FUNCTION_BLOCK PnpXYCalculator (* Composite Function Block Type *)
  (* Standard: 61499-2 *)
  (* Version 0.2, 2003-12-05, JHC, Rockwell Automation, Renamed from NEWCOMPFB. *)
  (* Version 0.1, 2002-01-08, JHC, Rockwell Automation, Added DLY FB as example. *)
  (* Version 0.0, 2000-05-27, JHC, Rockwell Automation *)
  (* Compiler header: package fb.rt.pnp; *)
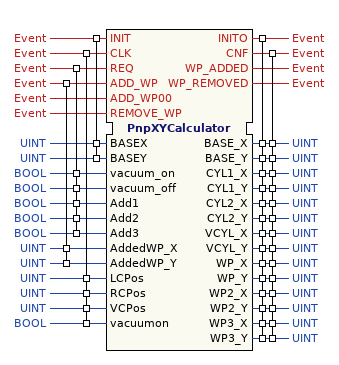
  EVENT_INPUT
    INIT WITH BASEX, BASEY; (* Initialization Request *)
    CLK WITH LCPos, RCPos, VCPos, vacuumon; (* Clock *)
    REQ WITH vacuum_on, vacuum_off, Add1, Add2, Add3;
    ADD_WP WITH AddedWP_X, AddedWP_Y;
    ADD_WP00;
    REMOVE_WP;
  END_EVENT
  EVENT_OUTPUT
    INITO WITH CYL1_X, CYL1_Y, BASE_Y, BASE_X, CYL2_X, CYL2_Y, VCYL_X, VCYL_Y, WP_X, WP_Y, WP2_X, WP2_Y, WP3_X, WP3_Y; (* Initialization Confirm *)
    CNF WITH CYL1_X, CYL1_Y, BASE_Y, BASE_X, CYL2_X, CYL2_Y, VCYL_X, VCYL_Y, WP_X, WP_Y, WP2_X, WP2_Y, WP3_X, WP3_Y;
    WP_ADDED;
    WP_REMOVED;
  END_EVENT
  VAR_INPUT
    BASEX : UINT;
    BASEY : UINT;
    vacuum_on : BOOL;
    vacuum_off : BOOL;
    Add1 : BOOL;
    Add2 : BOOL;
    Add3 : BOOL;
    AddedWP_X : UINT;
    AddedWP_Y : UINT;
    LCPos : UINT;
    RCPos : UINT;
    VCPos : UINT;
    vacuumon : BOOL;
  END_VAR
  VAR_OUTPUT
    BASE_X : UINT; (* Response Data from Socket *)
    BASE_Y : UINT; (* Response Data from Socket *)
    CYL1_X : UINT; (* Response Data from Socket *)
    CYL1_Y : UINT; (* Response Data from Socket *)
    CYL2_X : UINT; (* Response Data from Socket *)
    CYL2_Y : UINT; (* Response Data from Socket *)
    VCYL_X : UINT; (* Response Data from Socket *)
    VCYL_Y : UINT; (* Response Data from Socket *)
    WP_X : UINT; (* Response Data from Socket *)
    WP_Y : UINT; (* Response Data from Socket *)
    WP2_X : UINT; (* Response Data from Socket *)
    WP2_Y : UINT; (* Response Data from Socket *)
    WP3_X : UINT; (* Response Data from Socket *)
    WP3_Y : UINT; (* Response Data from Socket *)
  END_VAR
  VAR
    cyl1x : UINT;
    cyl2x : UINT;
    vcyly : UINT;
    wpx : UINT;
    wpy : UINT;
    wp2x : UINT;
    wp2y : UINT;
    wp3x : UINT;
    wp3y : UINT;
    slider1 : BOOL;
    slider2 : BOOL;
    slider3 : BOOL;
    wpon : BOOL;
    wp2on : BOOL;
    wp3on : BOOL;
  END_VAR
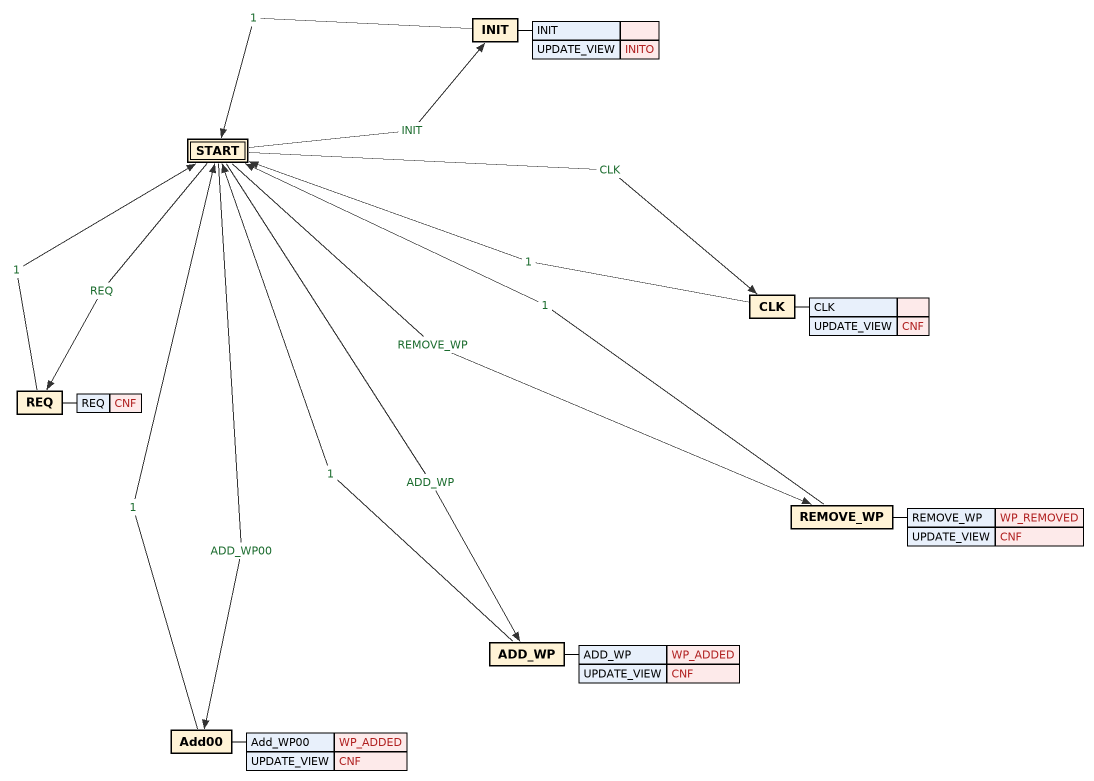
  EC_STATES
    START; (* Initial State *)
    INIT : INIT, UPDATE_VIEW -> INITO; (* Initialization *)
    REQ : REQ -> CNF; (* Normal execution *)
    CLK : CLK, UPDATE_VIEW -> CNF;
    ADD_WP : ADD_WP -> WP_ADDED, UPDATE_VIEW -> CNF;
    REMOVE_WP : REMOVE_WP -> WP_REMOVED, UPDATE_VIEW -> CNF;
    Add00 : Add_WP00 -> WP_ADDED, UPDATE_VIEW -> CNF;
  END_STATES
  EC_TRANSITIONS
    START TO INIT := INIT;
    INIT TO START := 1;
    START TO REQ := REQ;
    REQ TO START := 1;
    START TO CLK := CLK;
    CLK TO START := 1;
    START TO ADD_WP := ADD_WP;
    ADD_WP TO START := 1;
    START TO REMOVE_WP := REMOVE_WP;
    REMOVE_WP TO START := 1;
    START TO Add00 := ADD_WP00;
    Add00 TO START := 1;
  END_TRANSITIONS
  ALGORITHM INIT IN Java: (* Initialization algorithm *)
wpx.value = 6000;
wpy.value = 6000;
wp2x.value = 6000;
wp2y.value = 6000;
wp3x.value = 6000;
wp3y.value = 6000;
wpon.value = false;
wp2on.value = false;
wp3on.value = false;

BASE_X.value = BASEX.value;
BASE_Y.value = BASEY.value;
CYL1_Y.value = BASEY.value;
CYL2_Y.value = BASEY.value+12;
  END_ALGORITHM
  ALGORITHM REQ IN Java: (* Normally executed algorithm *)

  END_ALGORITHM
  ALGORITHM CLK IN Java:
int cyl1_length = 75;
int cyl2_length = 150;
int vcyl_length = 75;

// horizontal cylinder 1
cyl1x.value = LCPos.value;

// horizontal cylinder 2
cyl2x.value = RCPos.value;

// vertical cylinder
vcyly.value = VCPos.value;

if(wpx.value<=10 && wpy.value>=185){
slider1.value=true;
} else {slider1.value=false;}
if(wp2x.value<=10 && wp2y.value>=185){
slider2.value=true;
} else {slider2.value=false;}
if(wp3x.value<=10 && wp3y.value>=185){
slider3.value=true;
} else {slider3.value=false;}

if (vacuumon.value) {
int vacuumx = cyl1x.value+cyl2x.value;
int vacuumy = vcyly.value+115;
int dx = Math.abs(wpx.value - vacuumx);
int dy = Math.abs(wpy.value-vacuumy);
int dx2 = Math.abs(wp2x.value - vacuumx);
int dy2 = Math.abs(wp2y.value-vacuumy);
int dx3 = Math.abs(wp3x.value - vacuumx);
int dy3 = Math.abs(wp3y.value-vacuumy);

if (dx < 17 && dy < 7 && wp2on.value==false && wp3on.value==false){
wpon.value = true;
}
if (dx2 < 17 && dy2 < 7 && wpon.value==false && wp3on.value==false){
wp2on.value = true;
}
if (dx3 < 17 && dy3 < 7 && wp2on.value==false && wpon.value==false){
wp3on.value = true;
}
} else {
wpon.value = false;
wp2on.value = false;
wp3on.value = false;
}

//System.out.println("Clocking");
  END_ALGORITHM
  ALGORITHM UPDATE_VIEW IN Java:
int bx = BASEX.value;
int by = BASEY.value;
CYL1_X.value = bx+22+cyl1x.value;
CYL2_X.value = bx+116+cyl1x.value+cyl2x.value;
VCYL_X.value = bx+305+cyl1x.value+cyl2x.value;
VCYL_Y.value = by+vcyly.value+15;

if (wpon.value){
wpx.value = cyl1x.value+cyl2x.value;
wpy.value = vcyly.value+115;
} else if (slider1.value){
wpy.value = wpy.value+1;
} else {
wpy.value = 190;
}
if (wp2on.value){
wp2x.value = cyl1x.value+cyl2x.value;
wp2y.value = vcyly.value+115;
} else if (slider2.value){
wp2y.value = wp2y.value+1;
}else {
wp2y.value = 190;
}
if (wp3on.value){
wp3x.value = cyl1x.value+cyl2x.value;
wp3y.value = vcyly.value+115;
} else if (slider3.value){
wp3y.value = wp3y.value+1;
}else {
wp3y.value = 190;
}

WP_X.value = bx+300+wpx.value;
WP_Y.value = by+wpy.value;
WP2_X.value = bx+300+wp2x.value;
WP2_Y.value = by+wp2y.value;
WP3_X.value = bx+300+wp3x.value;
WP3_Y.value = by+wp3y.value;
if (WP_X.value == 305 && WP_Y.value >= 330)
{
    WP_X.value = 6000;
    WP_Y.value = 6000;
}
if (WP2_X.value == 305 && WP2_Y.value >= 330)
{
    WP2_X.value = 6000;
    WP2_Y.value = 6000;
}
if (WP3_X.value == 305 && WP3_Y.value >= 330)
{
    WP3_X.value = 6000;
    WP3_Y.value = 6000;
}

//System.out.println("C1X = " + CYL1_X + " C2X = " + CYL2_X + " VCX = " + VCYL_X + " VCY = " + VCYL_Y);
  END_ALGORITHM
  ALGORITHM ADD_WP IN Java:
if (Add1.value==true) {
wpx.value = 75;
wpy.value = 215;
wpon.value = false;
}
if (Add2.value==true) {
wp2x.value = 150;
wp2y.value = 215;
wp2on.value = false;
}
if (Add3.value==true) {
wp3x.value = 225;
wp3y.value = 215;
wp3on.value = false;
}
  END_ALGORITHM
  ALGORITHM REMOVE_WP IN Java:
if (Add1.value==true) {
wpon.value = false;
wpx.value = 6000;
wpy.value = 6000;
}
if (Add2.value==true) {
wp2on.value = false;
wp2x.value = 6000;
wp2y.value = 6000;
}
if (Add3.value==true) {
wp3on.value = false;
wp3x.value = 6000;
wp3y.value = 6000;
}
  END_ALGORITHM
  ALGORITHM Add_WP00 IN Java:
if (Add1.value==true) {
wpx.value = 0;
wpy.value = 215;
wpon.value = false;
}
if (Add2.value==true) {
wp2x.value = 0;
wp2y.value = 215;
wp2on.value = false;
}
if (Add3.value==true) {
wp3x.value = 0;
wp3y.value = 215;
wp3on.value = false;
}
  END_ALGORITHM
END_FUNCTION_BLOCK
